% RSLogix 500 project test.RSS, saved by version 8.30.00.16 %
PROJECT "UNTITLED"    % processor: Bul.1763 MicroLogix 1100 Series B %

PROGRAM FILES
  LAD 2   7 rungs

DATA FILES
  O0 OUTPUT  4 elements
  I1 INPUT  6 elements
  S2 STATUS  66 elements
  B3 BINARY  1 elements
  T4 TIMER  1 elements
  C5 COUNTER  1 elements
  R6 CONTROL  1 elements
  N7 INTEGER  1 elements
  F8 FLOAT  1 elements

LADDER 2
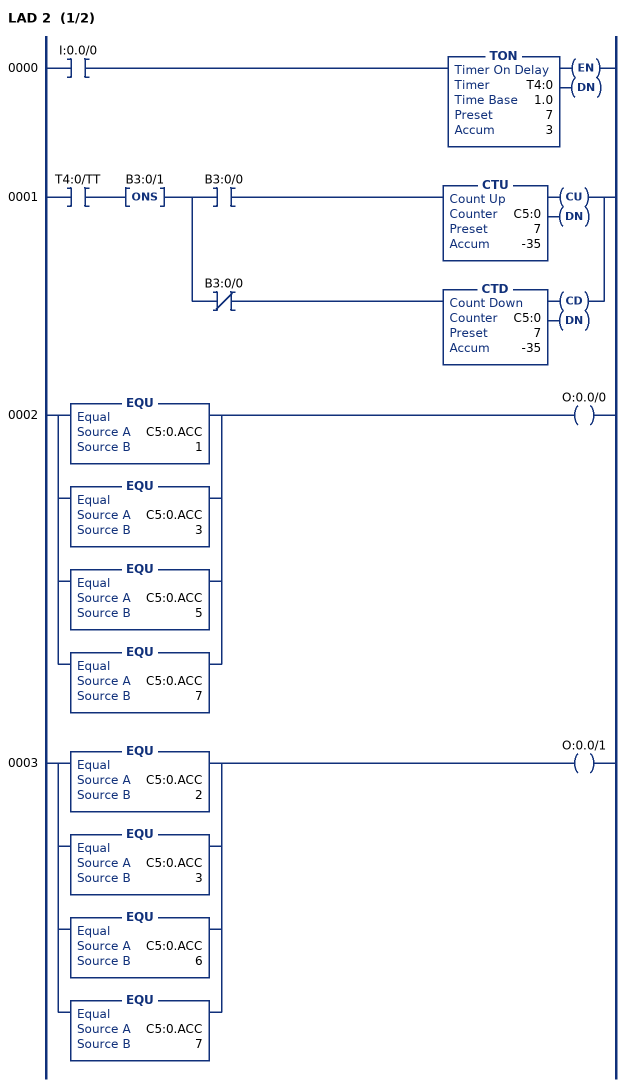
% Rung: 0 %
SOR XIC I:0.0/0 TON T4:0 1.0 7 3 EOR
% Rung: 1 %
SOR XIC T4:0/TT ONS B3:0/1 BST XIC B3:0/0 CTU C5:0 7 -35 NXB XIO B3:0/0 CTD C5:0 7 -35 BND EOR
% Rung: 2 %
SOR BST EQU C5:0.ACC 1 NXB EQU C5:0.ACC 3 NXB EQU C5:0.ACC 5 NXB EQU C5:0.ACC 7 BND OTE O:0.0/0 EOR
% Rung: 3 %
SOR BST EQU C5:0.ACC 2 NXB EQU C5:0.ACC 3 NXB EQU C5:0.ACC 6 NXB EQU C5:0.ACC 7 BND OTE O:0.0/1 EOR

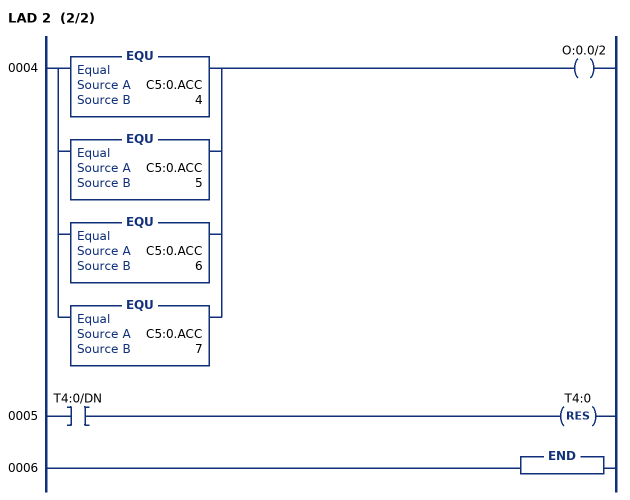
% Rung: 4 %
SOR BST EQU C5:0.ACC 4 NXB EQU C5:0.ACC 5 NXB EQU C5:0.ACC 6 NXB EQU C5:0.ACC 7 BND OTE O:0.0/2 EOR
% Rung: 5 %
SOR XIC T4:0/DN RES T4:0 EOR
% Rung: 6 %
SOR END EOR

DATA TABLE (non-zero values as saved)
DATA B3
% B3:0 % 0X0002
DATA T4
% .PRE .ACC %
% T4:0 % 7 4
DATA C5
% .PRE .ACC %
% C5:0 % 7 -35
DATA N7
% N7:0 % 7
